FUNCTION_BLOCK ByteArrayComparer EXTENDS Object IMPLEMENTS IComparer
VAR
	_ClassName : STRING := __POUNAME();
END_VAR

{attribute 'monitoring' := 'call'}
PROPERTY ClassName : STRING
GET
ClassName := _ClassName;
END_GET
END_PROPERTY

{attribute "object_name" := "Compare"}
METHOD Compare : COMPARISION_RESULT
VAR_INPUT
	left : GENERIC_VALUE;
	right : GENERIC_VALUE;
END_VAR
VAR
	leftPointer : POINTER TO BYTE; 
	rightPointer : POINTER TO BYTE; 
	
	i : LINT;
END_VAR
IF left.Address = 0 AND right.Address = 0 THEN
	Compare := COMPARISION_RESULT.EQUALS;
	RETURN;
END_IF

IF left.Address = 0 THEN
	Compare := COMPARISION_RESULT.LEFT_LESS_RIGHT;
	RETURN;	
END_IF

IF right.Address = 0 THEN
	Compare := COMPARISION_RESULT.LEFT_GREATER_RIGHT;
	RETURN;	
END_IF

FOR i := 0 TO TO_LINT(MIN(left.Size, right.Size)) - 1 DO
	leftPointer := left.Address + TO_LWORD(i);
	rightPointer := right.Address + TO_LWORD(i);
	
	IF leftPointer^ < rightPointer^ THEN
		Compare := COMPARISION_RESULT.LEFT_LESS_RIGHT;
		RETURN;
	ELSIF leftPointer^ > rightPointer^ THEN
		Compare := COMPARISION_RESULT.LEFT_GREATER_RIGHT;
		RETURN;
	END_IF	
END_FOR

IF left.Size < right.Size THEN
	Compare := COMPARISION_RESULT.LEFT_LESS_RIGHT;
ELSIF left.Size > right.Size THEN
	Compare := COMPARISION_RESULT.LEFT_GREATER_RIGHT;
ELSE
	Compare := COMPARISION_RESULT.EQUALS;
END_IF
END_METHOD

{attribute 'monitoring' := 'call'}
PROPERTY Size : ULINT
GET
Size := XSIZEOF(THIS^);
END_GET
END_PROPERTY

END_FUNCTION_BLOCK

(* stored: Version 1.1.0.1
   POU ByteArrayComparer: Id {2bb53bb7-7d07-4a7a-896e-016e853fd868}, SpecialFunc None
   Property ClassName: Id {cf39d53b-ed13-4edf-ad55-696c13de665b}
   Get Get: Id {d30e6779-120e-49c2-abe1-17cbfac7965e}
   Method Compare: Id {ee7448b3-b623-4697-a6c8-19f6c43d07cb}
   Property Size: Id {b1a1240f-8b51-48b9-84a3-3c39c9b5cd85}
   Get Get: Id {7cf65b52-2f9d-4aa5-9cb0-fb0f5d03a50d} *)
